Staubli VAL3: find.pgx

public program find(string& x_sItem[], bool& x_bFound[])
  local num l_nIndex
  local num l_nOperator
  local num l_nValue
  local string l_sItem[2]
begin
  // REMOVE THE COUNT
  x_sItem=right(x_sItem,len(x_sItem)-len("NUM "))
  // look inside
  x_bFound=isDefined(saveInOut:cCount[x_sItem])
  if !x_bFound
    x_bFound=isDefined(saveInOut:aCount[x_sItem])
  endIf
end
